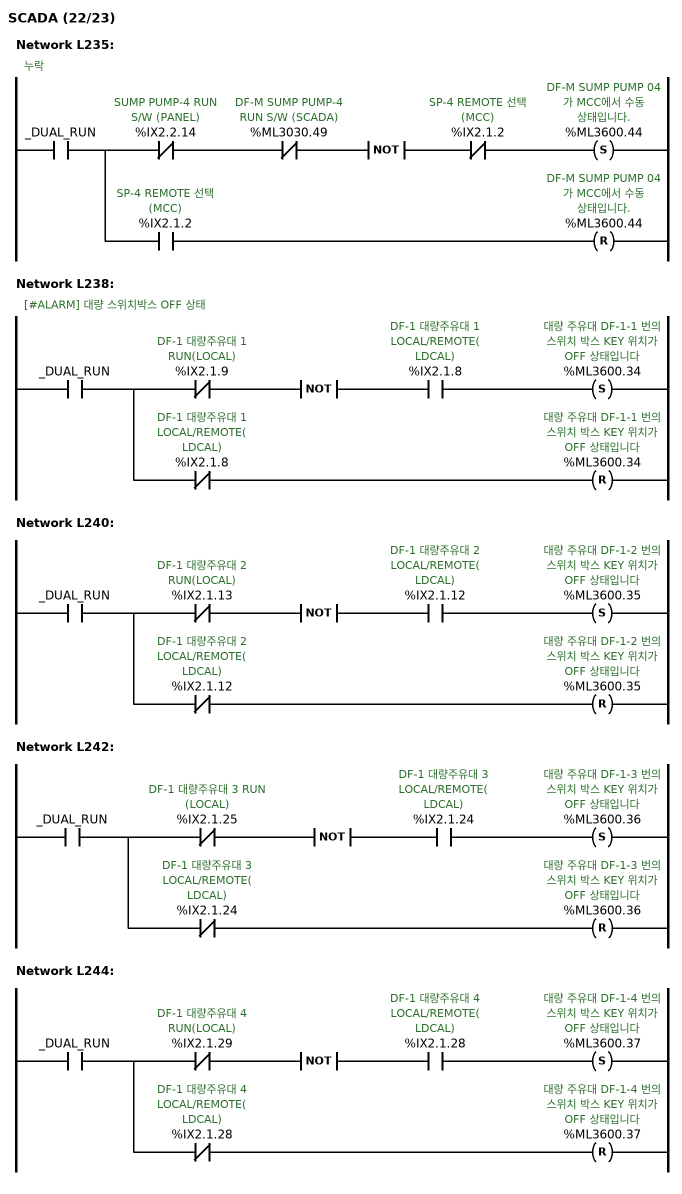
(* [picture p72: SCADA rungs L235-L244] *)
(* Rung L235 *)
IF NOT (_DUAL_RUN AND NOT %IX2.2.14 AND NOT %ML3030.49) AND NOT %IX2.1.2 THEN %ML3600.44 := TRUE; END_IF;
IF _DUAL_RUN AND %IX2.1.2 THEN %ML3600.44 := FALSE; END_IF;
(* 누락 *)
(* [#ALARM] 대량 스위치박스 OFF 상태 *)
(* Rung L238 *)
IF NOT (_DUAL_RUN AND NOT %IX2.1.9) AND %IX2.1.8 THEN %ML3600.34 := TRUE; END_IF;
IF _DUAL_RUN AND NOT %IX2.1.8 THEN %ML3600.34 := FALSE; END_IF;
(* Rung L240 *)
IF NOT (_DUAL_RUN AND NOT %IX2.1.13) AND %IX2.1.12 THEN %ML3600.35 := TRUE; END_IF;
IF _DUAL_RUN AND NOT %IX2.1.12 THEN %ML3600.35 := FALSE; END_IF;
(* Rung L242 *)
IF NOT (_DUAL_RUN AND NOT %IX2.1.25) AND %IX2.1.24 THEN %ML3600.36 := TRUE; END_IF;
IF _DUAL_RUN AND NOT %IX2.1.24 THEN %ML3600.36 := FALSE; END_IF;
(* Rung L244 *)
IF NOT (_DUAL_RUN AND NOT %IX2.1.29) AND %IX2.1.28 THEN %ML3600.37 := TRUE; END_IF;
IF _DUAL_RUN AND NOT %IX2.1.28 THEN %ML3600.37 := FALSE; END_IF;

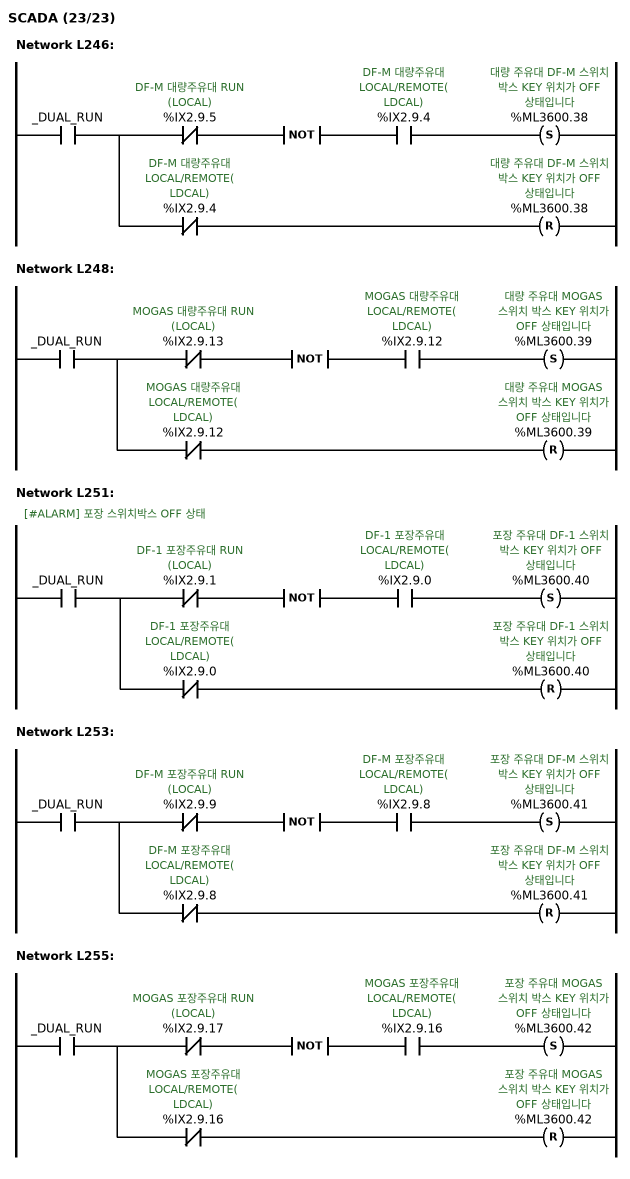
(* Rung L246 *)
IF NOT (_DUAL_RUN AND NOT %IX2.9.5) AND %IX2.9.4 THEN %ML3600.38 := TRUE; END_IF;
IF _DUAL_RUN AND NOT %IX2.9.4 THEN %ML3600.38 := FALSE; END_IF;
(* Rung L248 *)
IF NOT (_DUAL_RUN AND NOT %IX2.9.13) AND %IX2.9.12 THEN %ML3600.39 := TRUE; END_IF;
IF _DUAL_RUN AND NOT %IX2.9.12 THEN %ML3600.39 := FALSE; END_IF;
(* [#ALARM] 포장 스위치박스 OFF 상태 *)
(* Rung L251 *)
IF NOT (_DUAL_RUN AND NOT %IX2.9.1) AND %IX2.9.0 THEN %ML3600.40 := TRUE; END_IF;
IF _DUAL_RUN AND NOT %IX2.9.0 THEN %ML3600.40 := FALSE; END_IF;
(* Rung L253 *)
IF NOT (_DUAL_RUN AND NOT %IX2.9.9) AND %IX2.9.8 THEN %ML3600.41 := TRUE; END_IF;
IF _DUAL_RUN AND NOT %IX2.9.8 THEN %ML3600.41 := FALSE; END_IF;
(* Rung L255 *)
IF NOT (_DUAL_RUN AND NOT %IX2.9.17) AND %IX2.9.16 THEN %ML3600.42 := TRUE; END_IF;
IF _DUAL_RUN AND NOT %IX2.9.16 THEN %ML3600.42 := FALSE; END_IF;
END_PROGRAM

PROGRAM OUT (* task: 스캔 프로그램 *)
VAR
    D10 : BOOL;
    D1000 : BOOL;
    H16 : BOOL;
    INST : FF;
END_VAR
VAR
    _t1 : BOOL;
    _t2 : BOOL;
    _t3 : BOOL;
    _t4 : BOOL;
    _t5 : BOOL;
    _t6 : BOOL;
    _t7 : BOOL;
    _t8 : BOOL;
    _t9 : BOOL;
    _t10 : BOOL;
    _t11 : BOOL;
    _t12 : BOOL;
END_VAR

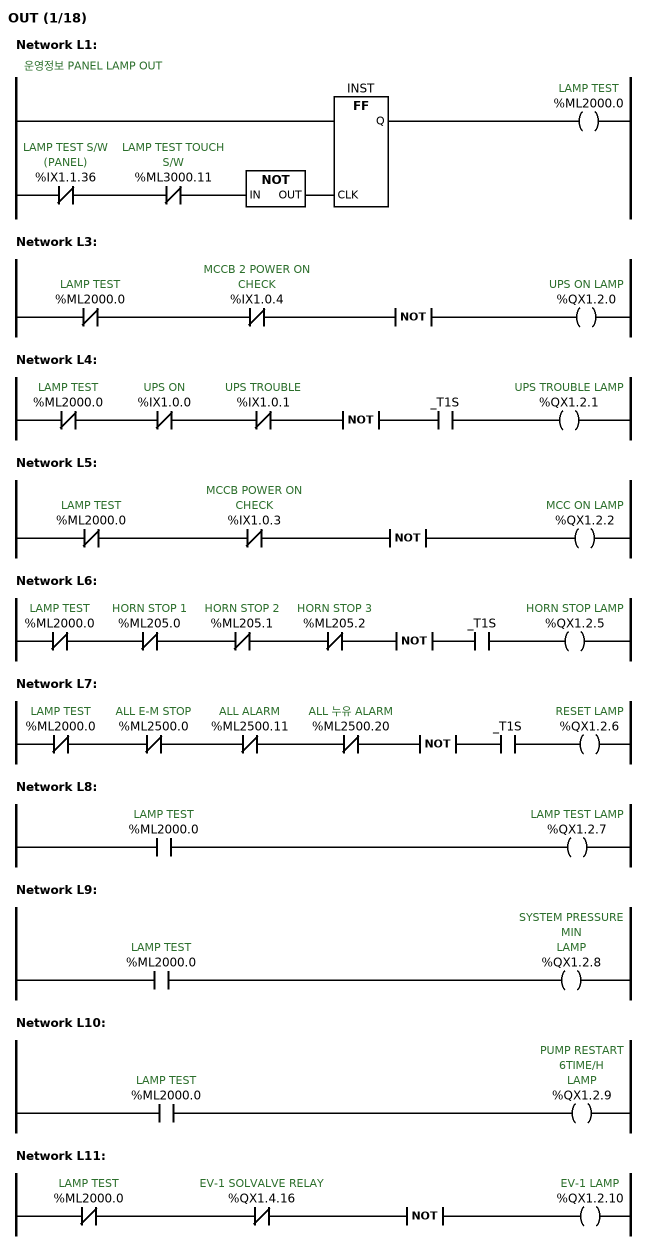
(* 운영정보 PANEL LAMP OUT *)
(* Rung L1 *)
INST(CLK := NOT (NOT %IX1.1.36 AND NOT %ML3000.11));
%ML2000.0 := INST.Q;
(* Rung L3 *)
%QX1.2.0 := NOT (NOT %ML2000.0 AND NOT %IX1.0.4);
(* Rung L4 *)
%QX1.2.1 := NOT (NOT %ML2000.0 AND NOT %IX1.0.0 AND NOT %IX1.0.1) AND _T1S;
(* Rung L5 *)
%QX1.2.2 := NOT (NOT %ML2000.0 AND NOT %IX1.0.3);
(* Rung L6 *)
%QX1.2.5 := NOT (NOT %ML2000.0 AND NOT %ML205.0 AND NOT %ML205.1 AND NOT %ML205.2) AND _T1S;
(* Rung L7 *)
%QX1.2.6 := NOT (NOT %ML2000.0 AND NOT %ML2500.0 AND NOT %ML2500.11 AND NOT %ML2500.20) AND _T1S;
(* Rung L8 *)
%QX1.2.7 := %ML2000.0;
(* Rung L9 *)
%QX1.2.8 := %ML2000.0;
(* Rung L10 *)
%QX1.2.9 := %ML2000.0;
(* Rung L11 *)
%QX1.2.10 := NOT (NOT %ML2000.0 AND NOT %QX1.4.16);

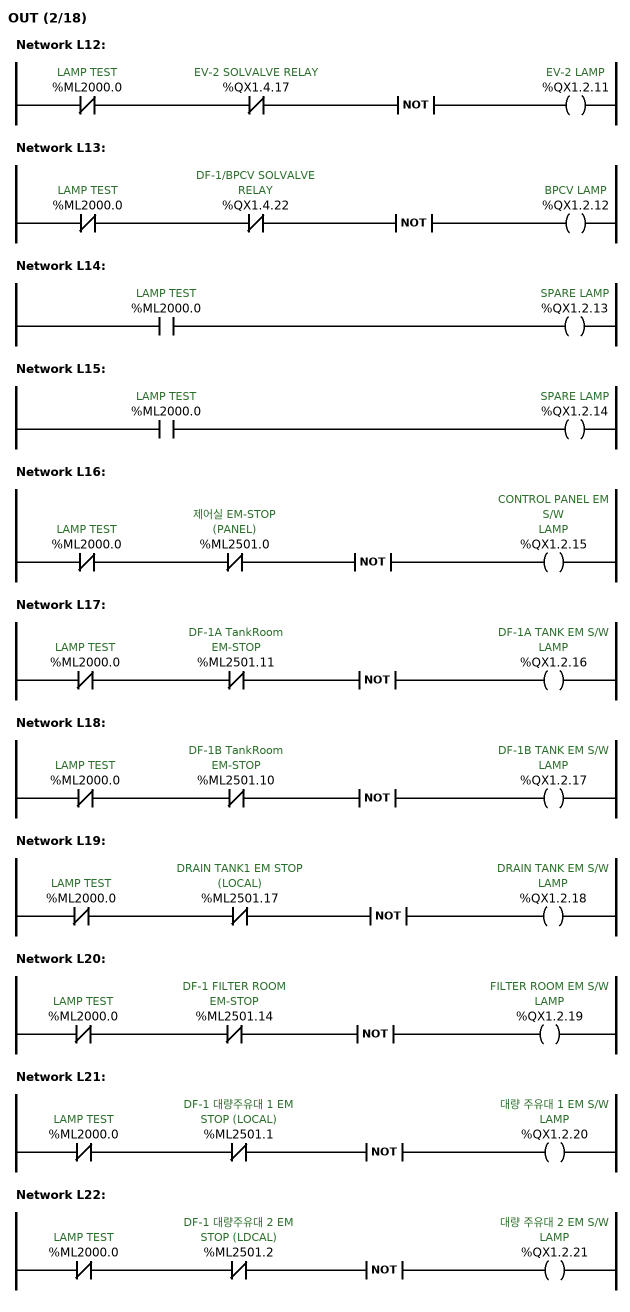
(* Rung L12 *)
%QX1.2.11 := NOT (NOT %ML2000.0 AND NOT %QX1.4.17);
(* Rung L13 *)
%QX1.2.12 := NOT (NOT %ML2000.0 AND NOT %QX1.4.22);
(* Rung L14 *)
%QX1.2.13 := %ML2000.0;
(* Rung L15 *)
%QX1.2.14 := %ML2000.0;
(* Rung L16 *)
%QX1.2.15 := NOT (NOT %ML2000.0 AND NOT %ML2501.0);
(* Rung L17 *)
%QX1.2.16 := NOT (NOT %ML2000.0 AND NOT %ML2501.11);
(* Rung L18 *)
%QX1.2.17 := NOT (NOT %ML2000.0 AND NOT %ML2501.10);
(* Rung L19 *)
%QX1.2.18 := NOT (NOT %ML2000.0 AND NOT %ML2501.17);
(* Rung L20 *)
%QX1.2.19 := NOT (NOT %ML2000.0 AND NOT %ML2501.14);
(* Rung L21 *)
%QX1.2.20 := NOT (NOT %ML2000.0 AND NOT %ML2501.1);
(* Rung L22 *)
%QX1.2.21 := NOT (NOT %ML2000.0 AND NOT %ML2501.2);

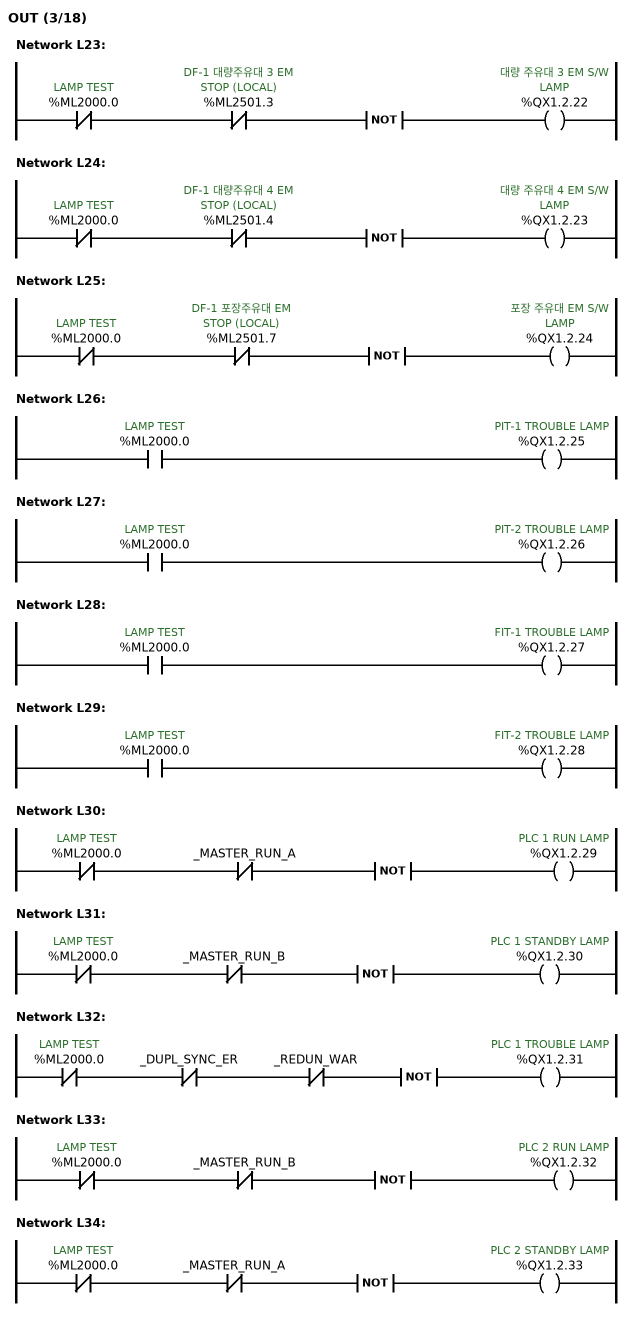
(* Rung L23 *)
%QX1.2.22 := NOT (NOT %ML2000.0 AND NOT %ML2501.3);
(* Rung L24 *)
%QX1.2.23 := NOT (NOT %ML2000.0 AND NOT %ML2501.4);
(* Rung L25 *)
%QX1.2.24 := NOT (NOT %ML2000.0 AND NOT %ML2501.7);
(* Rung L26 *)
%QX1.2.25 := %ML2000.0;
(* Rung L27 *)
%QX1.2.26 := %ML2000.0;
(* Rung L28 *)
%QX1.2.27 := %ML2000.0;
(* Rung L29 *)
%QX1.2.28 := %ML2000.0;
(* Rung L30 *)
%QX1.2.29 := NOT (NOT %ML2000.0 AND NOT _MASTER_RUN_A);
(* Rung L31 *)
%QX1.2.30 := NOT (NOT %ML2000.0 AND NOT _MASTER_RUN_B);
(* Rung L32 *)
%QX1.2.31 := NOT (NOT %ML2000.0 AND NOT _DUPL_SYNC_ER AND NOT _REDUN_WAR);
(* Rung L33 *)
%QX1.2.32 := NOT (NOT %ML2000.0 AND NOT _MASTER_RUN_B);
(* Rung L34 *)
%QX1.2.33 := NOT (NOT %ML2000.0 AND NOT _MASTER_RUN_A);

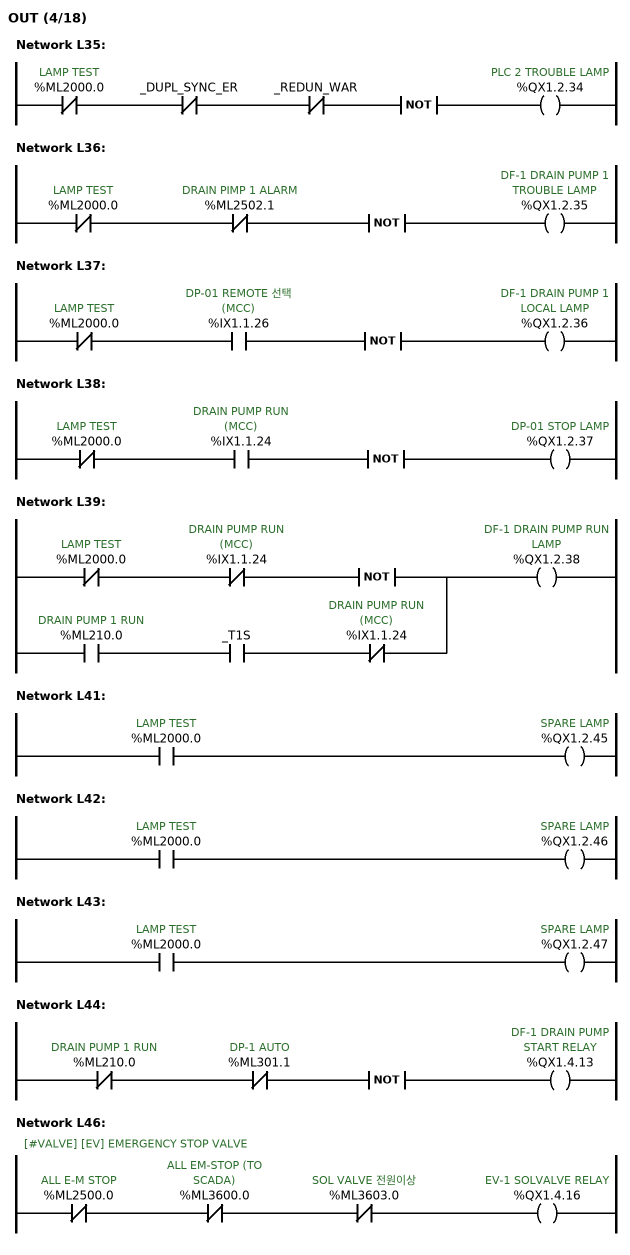
(* Rung L35 *)
%QX1.2.34 := NOT (NOT %ML2000.0 AND NOT _DUPL_SYNC_ER AND NOT _REDUN_WAR);
(* Rung L36 *)
%QX1.2.35 := NOT (NOT %ML2000.0 AND NOT %ML2502.1);
(* Rung L37 *)
%QX1.2.36 := NOT (NOT %ML2000.0 AND %IX1.1.26);
(* Rung L38 *)
%QX1.2.37 := NOT (NOT %ML2000.0 AND %IX1.1.24);
(* Rung L39 *)
%QX1.2.38 := NOT (NOT %ML2000.0 AND NOT %IX1.1.24) OR (%ML210.0 AND _T1S AND NOT %IX1.1.24);
(* Rung L41 *)
%QX1.2.45 := %ML2000.0;
(* Rung L42 *)
%QX1.2.46 := %ML2000.0;
(* Rung L43 *)
%QX1.2.47 := %ML2000.0;
(* Rung L44 *)
%QX1.4.13 := NOT (NOT %ML210.0 AND NOT %ML301.1);
(* [#VALVE] [EV] EMERGENCY STOP VALVE *)
(* Rung L46 *)
%QX1.4.16 := NOT %ML2500.0 AND NOT %ML3600.0 AND NOT %ML3603.0;

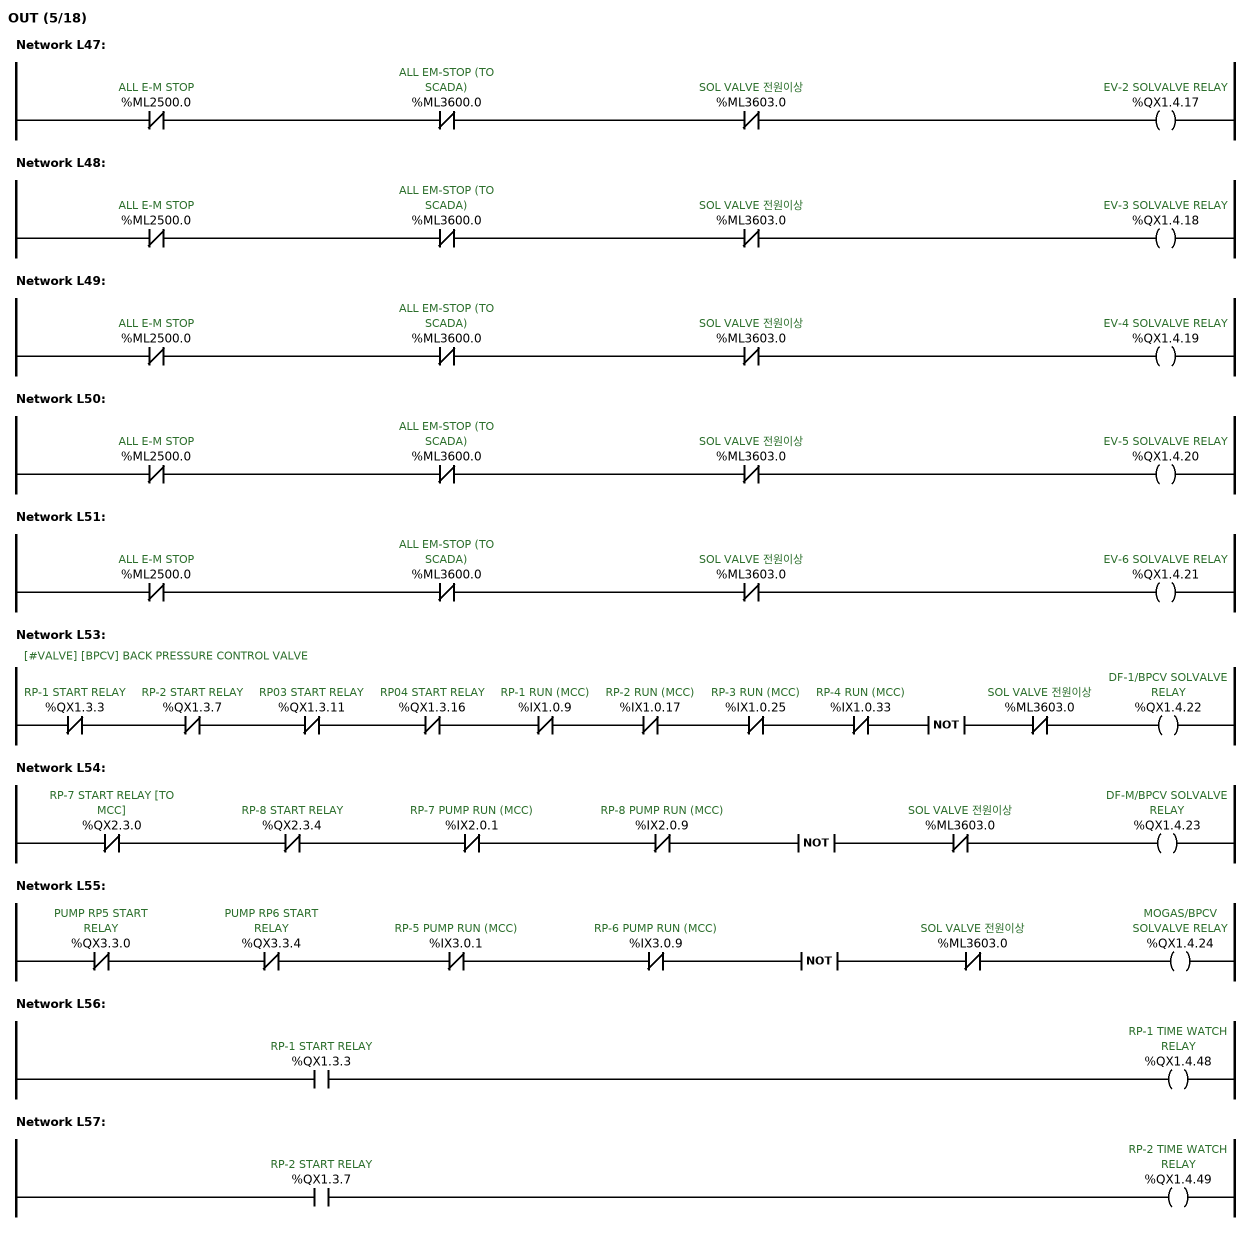
(* Rung L47 *)
%QX1.4.17 := NOT %ML2500.0 AND NOT %ML3600.0 AND NOT %ML3603.0;
(* Rung L48 *)
%QX1.4.18 := NOT %ML2500.0 AND NOT %ML3600.0 AND NOT %ML3603.0;
(* Rung L49 *)
%QX1.4.19 := NOT %ML2500.0 AND NOT %ML3600.0 AND NOT %ML3603.0;
(* Rung L50 *)
%QX1.4.20 := NOT %ML2500.0 AND NOT %ML3600.0 AND NOT %ML3603.0;
(* Rung L51 *)
%QX1.4.21 := NOT %ML2500.0 AND NOT %ML3600.0 AND NOT %ML3603.0;
(* [#VALVE] [BPCV] BACK PRESSURE CONTROL VALVE *)
(* Rung L53 *)
%QX1.4.22 := NOT (NOT %QX1.3.3 AND NOT %QX1.3.7 AND NOT %QX1.3.11 AND NOT %QX1.3.16 AND NOT %IX1.0.9 AND NOT %IX1.0.17 AND NOT %IX1.0.25 AND NOT %IX1.0.33) AND NOT %ML3603.0;
(* Rung L54 *)
%QX1.4.23 := NOT (NOT %QX2.3.0 AND NOT %QX2.3.4 AND NOT %IX2.0.1 AND NOT %IX2.0.9) AND NOT %ML3603.0;
(* Rung L55 *)
%QX1.4.24 := NOT (NOT %QX3.3.0 AND NOT %QX3.3.4 AND NOT %IX3.0.1 AND NOT %IX3.0.9) AND NOT %ML3603.0;
(* Rung L56 *)
%QX1.4.48 := %QX1.3.3;
(* Rung L57 *)
%QX1.4.49 := %QX1.3.7;

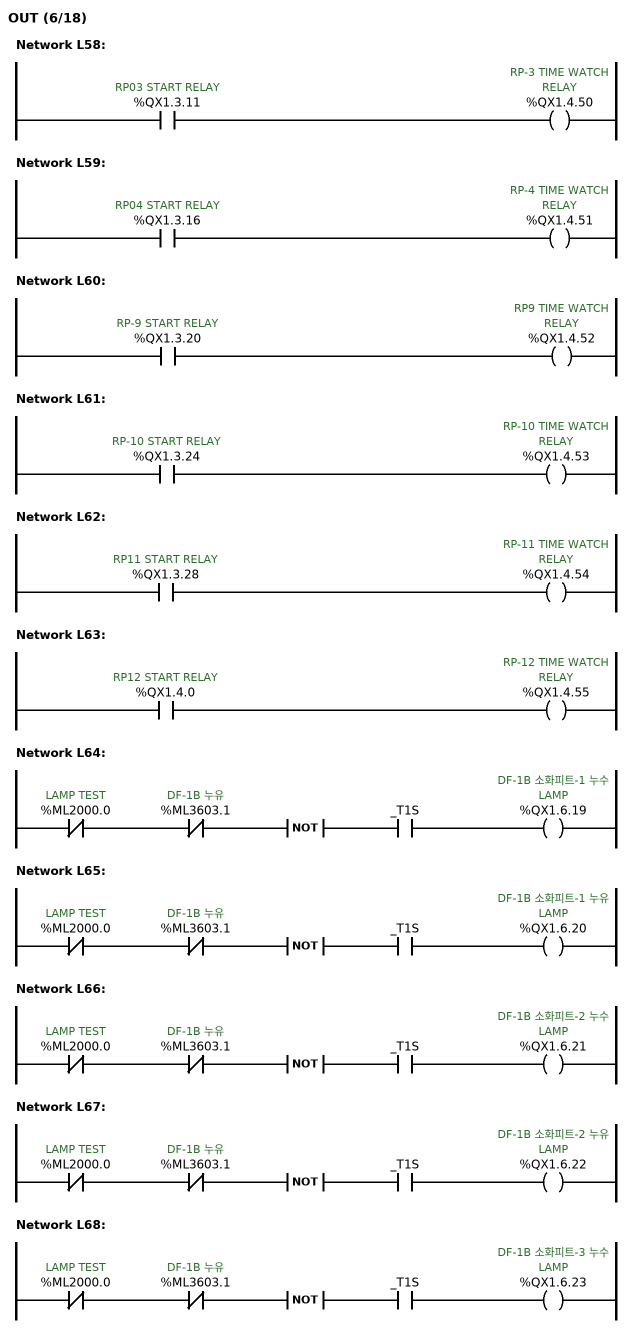
(* Rung L58 *)
%QX1.4.50 := %QX1.3.11;
(* Rung L59 *)
%QX1.4.51 := %QX1.3.16;
(* Rung L60 *)
%QX1.4.52 := %QX1.3.20;
(* Rung L61 *)
%QX1.4.53 := %QX1.3.24;
(* Rung L62 *)
%QX1.4.54 := %QX1.3.28;
(* Rung L63 *)
%QX1.4.55 := %QX1.4.0;
(* Rung L64 *)
%QX1.6.19 := NOT (NOT %ML2000.0 AND NOT %ML3603.1) AND _T1S;
(* Rung L65 *)
%QX1.6.20 := NOT (NOT %ML2000.0 AND NOT %ML3603.1) AND _T1S;
(* Rung L66 *)
%QX1.6.21 := NOT (NOT %ML2000.0 AND NOT %ML3603.1) AND _T1S;
(* Rung L67 *)
%QX1.6.22 := NOT (NOT %ML2000.0 AND NOT %ML3603.1) AND _T1S;
(* Rung L68 *)
%QX1.6.23 := NOT (NOT %ML2000.0 AND NOT %ML3603.1) AND _T1S;

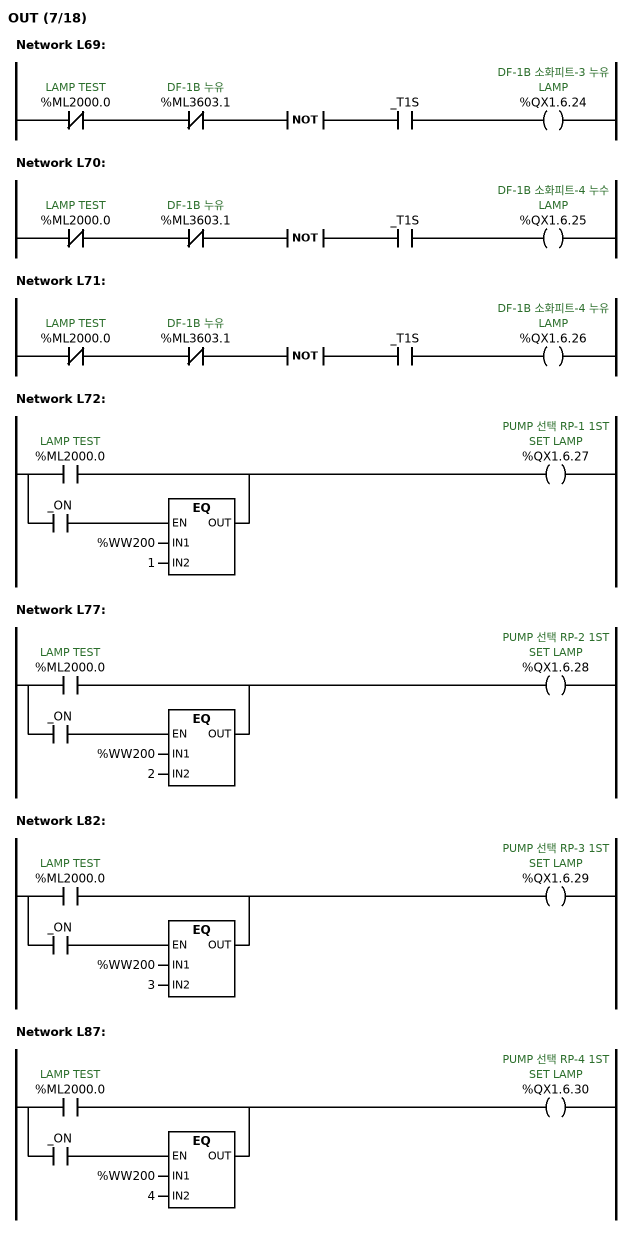
(* Rung L69 *)
%QX1.6.24 := NOT (NOT %ML2000.0 AND NOT %ML3603.1) AND _T1S;
(* Rung L70 *)
%QX1.6.25 := NOT (NOT %ML2000.0 AND NOT %ML3603.1) AND _T1S;
(* Rung L71 *)
%QX1.6.26 := NOT (NOT %ML2000.0 AND NOT %ML3603.1) AND _T1S;
(* Rung L72 *)
IF _ON THEN _t1 := %WW200 = 1; END_IF;
%QX1.6.27 := %ML2000.0 OR _t1;
(* Rung L77 *)
IF _ON THEN _t2 := %WW200 = 2; END_IF;
%QX1.6.28 := %ML2000.0 OR _t2;
(* Rung L82 *)
IF _ON THEN _t3 := %WW200 = 3; END_IF;
%QX1.6.29 := %ML2000.0 OR _t3;
(* Rung L87 *)
IF _ON THEN _t4 := %WW200 = 4; END_IF;
%QX1.6.30 := %ML2000.0 OR _t4;

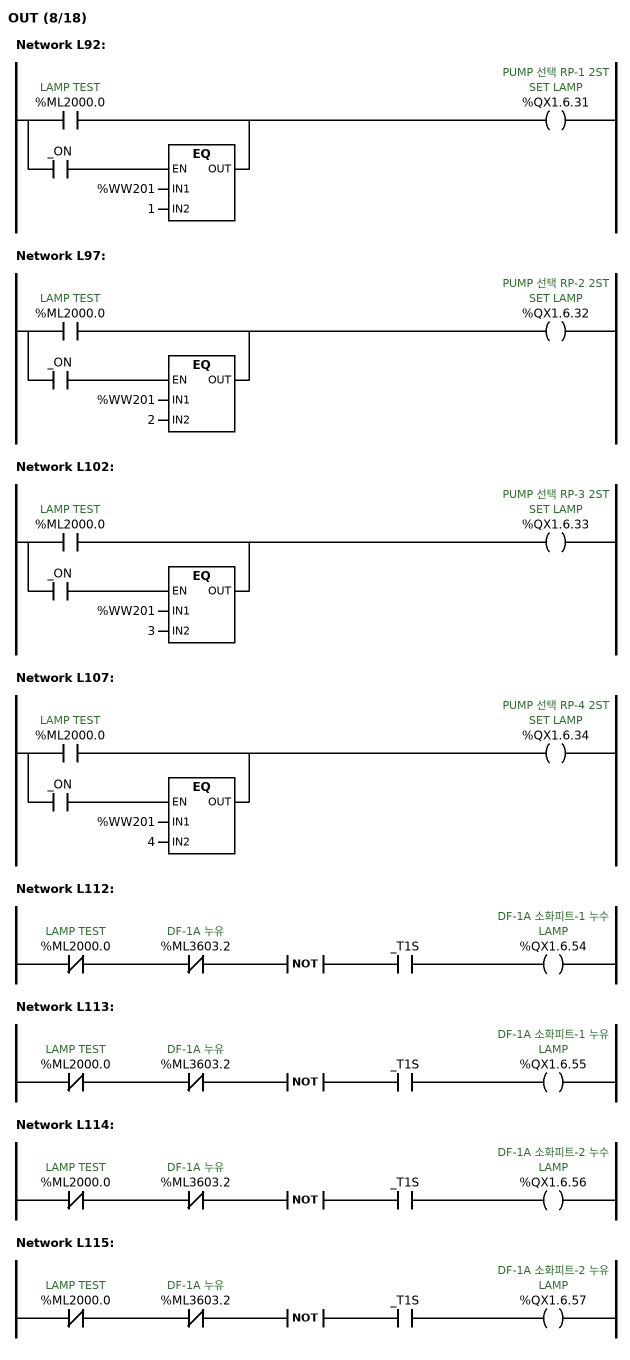
(* Rung L92 *)
IF _ON THEN _t5 := %WW201 = 1; END_IF;
%QX1.6.31 := %ML2000.0 OR _t5;
(* Rung L97 *)
IF _ON THEN _t6 := %WW201 = 2; END_IF;
%QX1.6.32 := %ML2000.0 OR _t6;
(* Rung L102 *)
IF _ON THEN _t7 := %WW201 = 3; END_IF;
%QX1.6.33 := %ML2000.0 OR _t7;
(* Rung L107 *)
IF _ON THEN _t8 := %WW201 = 4; END_IF;
%QX1.6.34 := %ML2000.0 OR _t8;
(* Rung L112 *)
%QX1.6.54 := NOT (NOT %ML2000.0 AND NOT %ML3603.2) AND _T1S;
(* Rung L113 *)
%QX1.6.55 := NOT (NOT %ML2000.0 AND NOT %ML3603.2) AND _T1S;
(* Rung L114 *)
%QX1.6.56 := NOT (NOT %ML2000.0 AND NOT %ML3603.2) AND _T1S;
(* Rung L115 *)
%QX1.6.57 := NOT (NOT %ML2000.0 AND NOT %ML3603.2) AND _T1S;

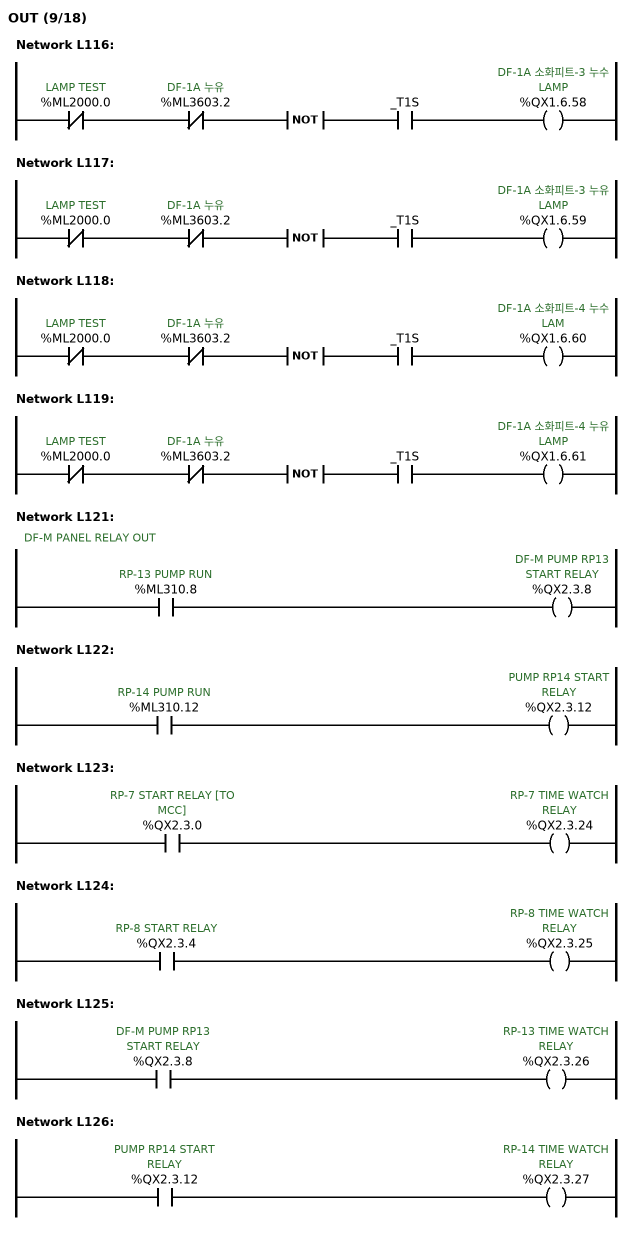
(* Rung L116 *)
%QX1.6.58 := NOT (NOT %ML2000.0 AND NOT %ML3603.2) AND _T1S;
(* Rung L117 *)
%QX1.6.59 := NOT (NOT %ML2000.0 AND NOT %ML3603.2) AND _T1S;
(* Rung L118 *)
%QX1.6.60 := NOT (NOT %ML2000.0 AND NOT %ML3603.2) AND _T1S;
(* Rung L119 *)
%QX1.6.61 := NOT (NOT %ML2000.0 AND NOT %ML3603.2) AND _T1S;
(* DF-M PANEL RELAY OUT *)
(* Rung L121 *)
%QX2.3.8 := %ML310.8;
(* Rung L122 *)
%QX2.3.12 := %ML310.12;
(* Rung L123 *)
%QX2.3.24 := %QX2.3.0;
(* Rung L124 *)
%QX2.3.25 := %QX2.3.4;
(* Rung L125 *)
%QX2.3.26 := %QX2.3.8;
(* Rung L126 *)
%QX2.3.27 := %QX2.3.12;

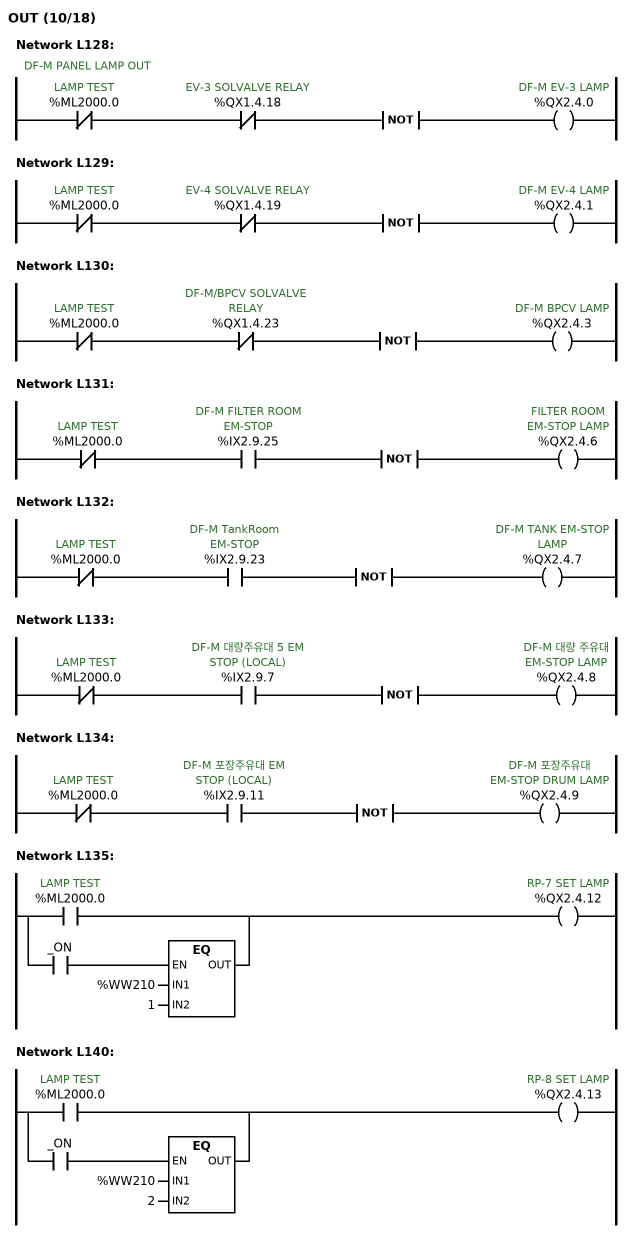
(* DF-M PANEL LAMP OUT *)
(* Rung L128 *)
%QX2.4.0 := NOT (NOT %ML2000.0 AND NOT %QX1.4.18);
(* Rung L129 *)
%QX2.4.1 := NOT (NOT %ML2000.0 AND NOT %QX1.4.19);
(* Rung L130 *)
%QX2.4.3 := NOT (NOT %ML2000.0 AND NOT %QX1.4.23);
(* Rung L131 *)
%QX2.4.6 := NOT (NOT %ML2000.0 AND %IX2.9.25);
(* Rung L132 *)
%QX2.4.7 := NOT (NOT %ML2000.0 AND %IX2.9.23);
(* Rung L133 *)
%QX2.4.8 := NOT (NOT %ML2000.0 AND %IX2.9.7);
(* Rung L134 *)
%QX2.4.9 := NOT (NOT %ML2000.0 AND %IX2.9.11);
(* Rung L135 *)
IF _ON THEN _t9 := %WW210 = 1; END_IF;
%QX2.4.12 := %ML2000.0 OR _t9;
(* Rung L140 *)
IF _ON THEN _t10 := %WW210 = 2; END_IF;
%QX2.4.13 := %ML2000.0 OR _t10;

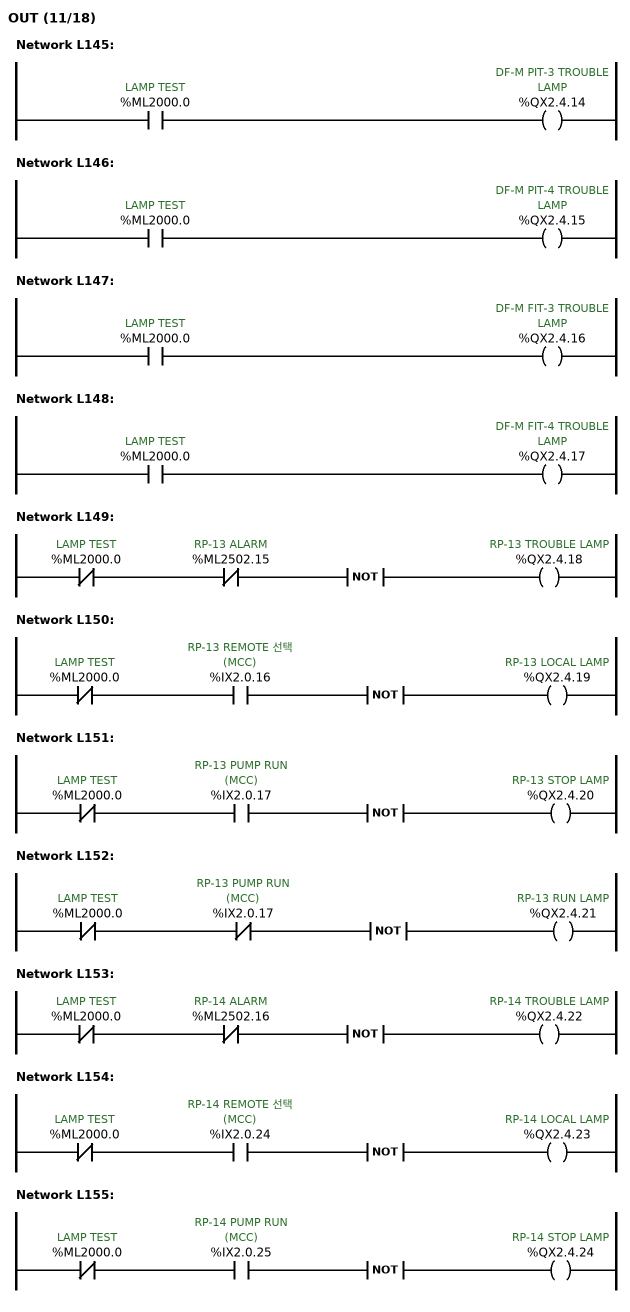
(* Rung L145 *)
%QX2.4.14 := %ML2000.0;
(* Rung L146 *)
%QX2.4.15 := %ML2000.0;
(* Rung L147 *)
%QX2.4.16 := %ML2000.0;
(* Rung L148 *)
%QX2.4.17 := %ML2000.0;
(* Rung L149 *)
%QX2.4.18 := NOT (NOT %ML2000.0 AND NOT %ML2502.15);
(* Rung L150 *)
%QX2.4.19 := NOT (NOT %ML2000.0 AND %IX2.0.16);
(* Rung L151 *)
%QX2.4.20 := NOT (NOT %ML2000.0 AND %IX2.0.17);
(* Rung L152 *)
%QX2.4.21 := NOT (NOT %ML2000.0 AND NOT %IX2.0.17);
(* Rung L153 *)
%QX2.4.22 := NOT (NOT %ML2000.0 AND NOT %ML2502.16);
(* Rung L154 *)
%QX2.4.23 := NOT (NOT %ML2000.0 AND %IX2.0.24);
(* Rung L155 *)
%QX2.4.24 := NOT (NOT %ML2000.0 AND %IX2.0.25);

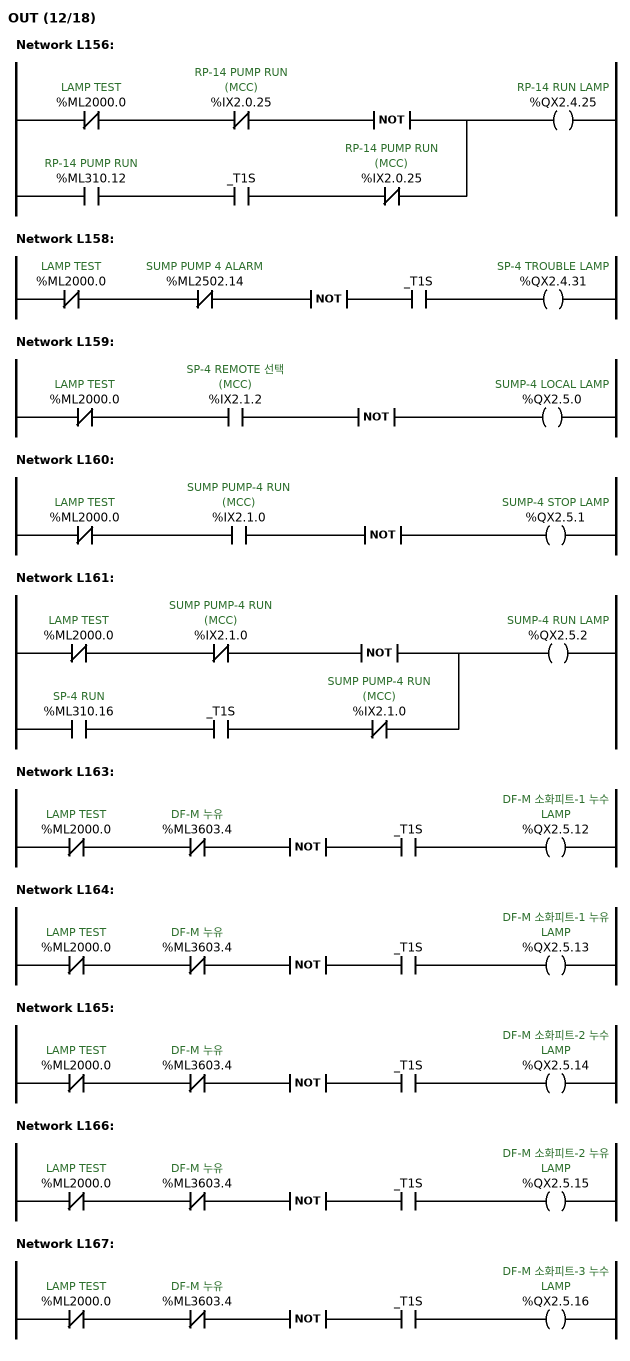
(* Rung L156 *)
%QX2.4.25 := NOT (NOT %ML2000.0 AND NOT %IX2.0.25) OR (%ML310.12 AND _T1S AND NOT %IX2.0.25);
(* Rung L158 *)
%QX2.4.31 := NOT (NOT %ML2000.0 AND NOT %ML2502.14) AND _T1S;
(* Rung L159 *)
%QX2.5.0 := NOT (NOT %ML2000.0 AND %IX2.1.2);
(* Rung L160 *)
%QX2.5.1 := NOT (NOT %ML2000.0 AND %IX2.1.0);
(* Rung L161 *)
%QX2.5.2 := NOT (NOT %ML2000.0 AND NOT %IX2.1.0) OR (%ML310.16 AND _T1S AND NOT %IX2.1.0);
(* Rung L163 *)
%QX2.5.12 := NOT (NOT %ML2000.0 AND NOT %ML3603.4) AND _T1S;
(* Rung L164 *)
%QX2.5.13 := NOT (NOT %ML2000.0 AND NOT %ML3603.4) AND _T1S;
(* Rung L165 *)
%QX2.5.14 := NOT (NOT %ML2000.0 AND NOT %ML3603.4) AND _T1S;
(* Rung L166 *)
%QX2.5.15 := NOT (NOT %ML2000.0 AND NOT %ML3603.4) AND _T1S;
(* Rung L167 *)
%QX2.5.16 := NOT (NOT %ML2000.0 AND NOT %ML3603.4) AND _T1S;

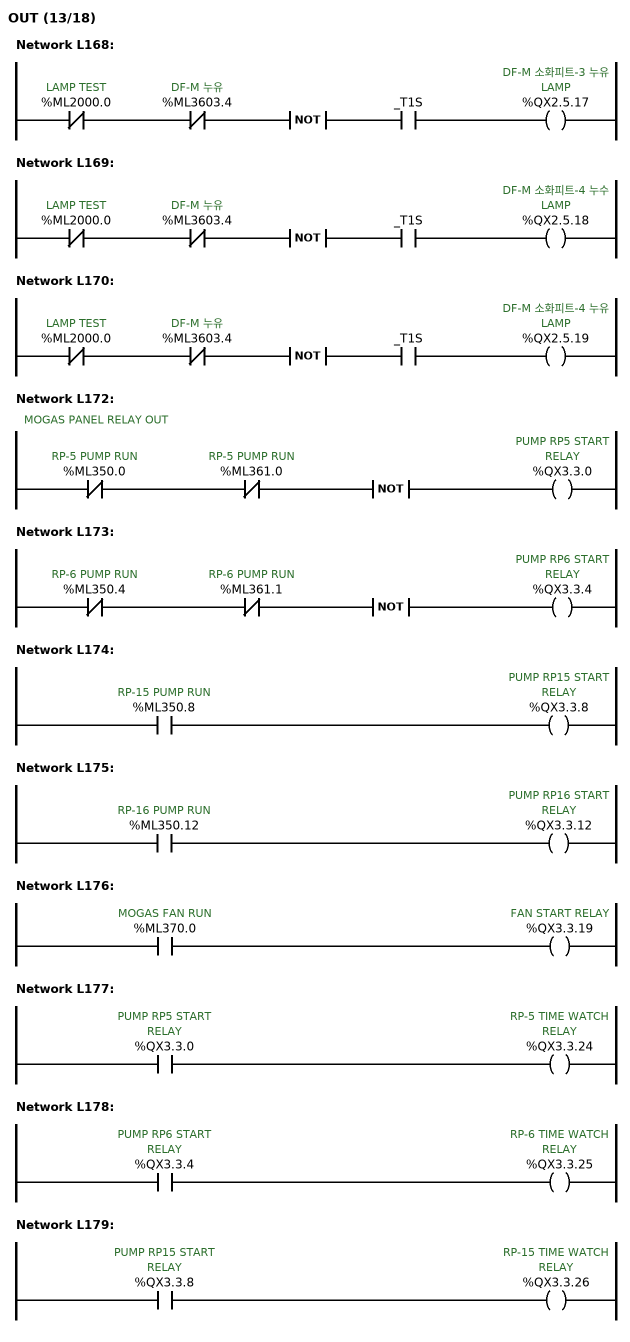
(* Rung L168 *)
%QX2.5.17 := NOT (NOT %ML2000.0 AND NOT %ML3603.4) AND _T1S;
(* Rung L169 *)
%QX2.5.18 := NOT (NOT %ML2000.0 AND NOT %ML3603.4) AND _T1S;
(* Rung L170 *)
%QX2.5.19 := NOT (NOT %ML2000.0 AND NOT %ML3603.4) AND _T1S;
(* MOGAS PANEL RELAY OUT *)
(* Rung L172 *)
%QX3.3.0 := NOT (NOT %ML350.0 AND NOT %ML361.0);
(* Rung L173 *)
%QX3.3.4 := NOT (NOT %ML350.4 AND NOT %ML361.1);
(* Rung L174 *)
%QX3.3.8 := %ML350.8;
(* Rung L175 *)
%QX3.3.12 := %ML350.12;
(* Rung L176 *)
%QX3.3.19 := %ML370.0;
(* Rung L177 *)
%QX3.3.24 := %QX3.3.0;
(* Rung L178 *)
%QX3.3.25 := %QX3.3.4;
(* Rung L179 *)
%QX3.3.26 := %QX3.3.8;

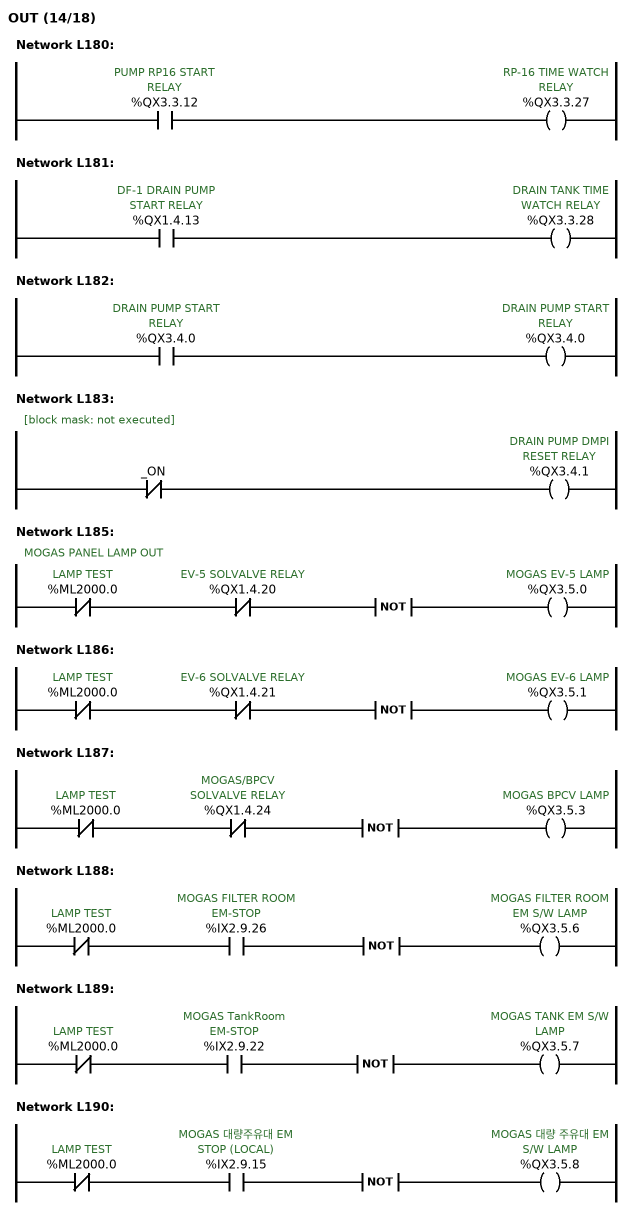
(* Rung L180 *)
%QX3.3.27 := %QX3.3.12;
(* Rung L181 *)
%QX3.3.28 := %QX1.4.13;
(* Rung L182 *)
%QX3.4.0 := %QX3.4.0;
(* Rung L183 is block-masked: not executed *)
// %QX3.4.1 := NOT _ON;
(* MOGAS PANEL LAMP OUT *)
(* Rung L185 *)
%QX3.5.0 := NOT (NOT %ML2000.0 AND NOT %QX1.4.20);
(* Rung L186 *)
%QX3.5.1 := NOT (NOT %ML2000.0 AND NOT %QX1.4.21);
(* Rung L187 *)
%QX3.5.3 := NOT (NOT %ML2000.0 AND NOT %QX1.4.24);
(* Rung L188 *)
%QX3.5.6 := NOT (NOT %ML2000.0 AND %IX2.9.26);
(* Rung L189 *)
%QX3.5.7 := NOT (NOT %ML2000.0 AND %IX2.9.22);
(* Rung L190 *)
%QX3.5.8 := NOT (NOT %ML2000.0 AND %IX2.9.15);

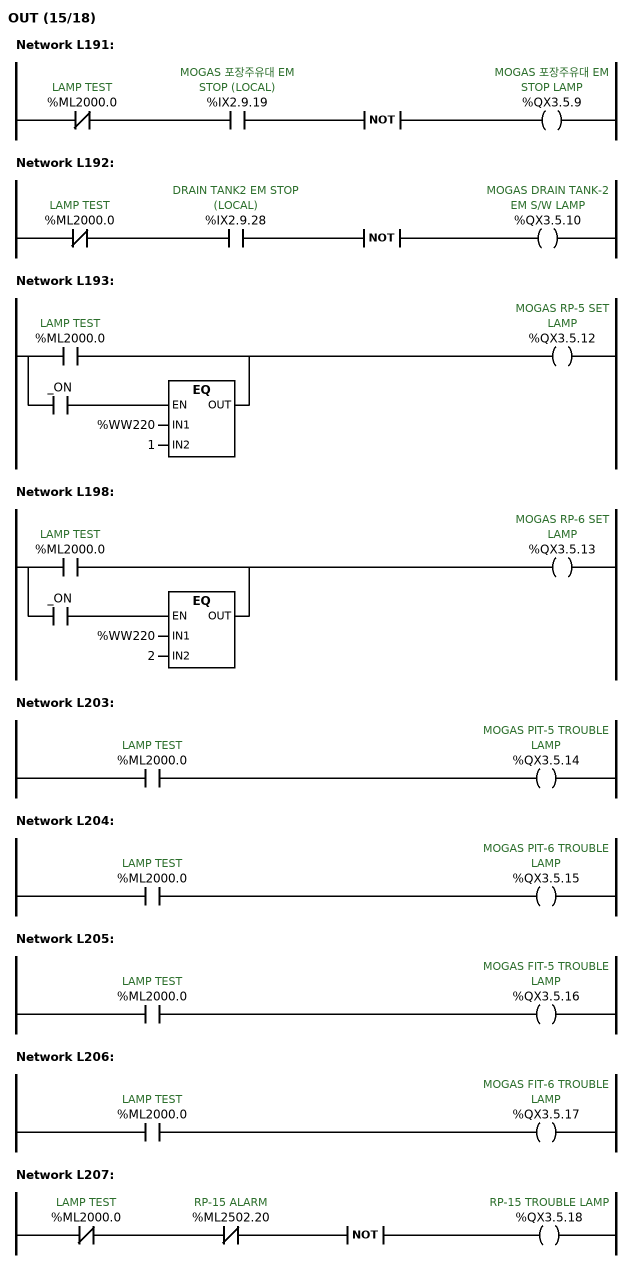
(* Rung L191 *)
%QX3.5.9 := NOT (NOT %ML2000.0 AND %IX2.9.19);
(* Rung L192 *)
%QX3.5.10 := NOT (NOT %ML2000.0 AND %IX2.9.28);
(* Rung L193 *)
IF _ON THEN _t11 := %WW220 = 1; END_IF;
%QX3.5.12 := %ML2000.0 OR _t11;
(* Rung L198 *)
IF _ON THEN _t12 := %WW220 = 2; END_IF;
%QX3.5.13 := %ML2000.0 OR _t12;
(* Rung L203 *)
%QX3.5.14 := %ML2000.0;
(* Rung L204 *)
%QX3.5.15 := %ML2000.0;
(* Rung L205 *)
%QX3.5.16 := %ML2000.0;
(* Rung L206 *)
%QX3.5.17 := %ML2000.0;
(* Rung L207 *)
%QX3.5.18 := NOT (NOT %ML2000.0 AND NOT %ML2502.20);

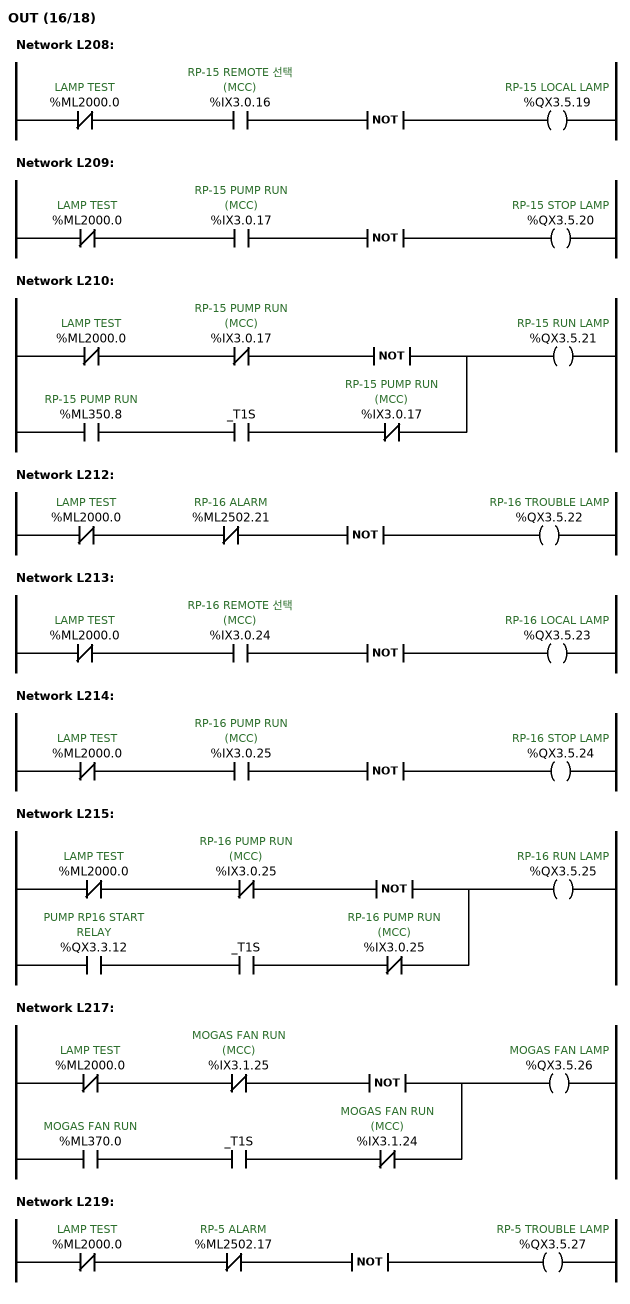
(* Rung L208 *)
%QX3.5.19 := NOT (NOT %ML2000.0 AND %IX3.0.16);
(* Rung L209 *)
%QX3.5.20 := NOT (NOT %ML2000.0 AND %IX3.0.17);
(* Rung L210 *)
%QX3.5.21 := NOT (NOT %ML2000.0 AND NOT %IX3.0.17) OR (%ML350.8 AND _T1S AND NOT %IX3.0.17);
(* Rung L212 *)
%QX3.5.22 := NOT (NOT %ML2000.0 AND NOT %ML2502.21);
(* Rung L213 *)
%QX3.5.23 := NOT (NOT %ML2000.0 AND %IX3.0.24);
(* Rung L214 *)
%QX3.5.24 := NOT (NOT %ML2000.0 AND %IX3.0.25);
(* Rung L215 *)
%QX3.5.25 := NOT (NOT %ML2000.0 AND NOT %IX3.0.25) OR (%QX3.3.12 AND _T1S AND NOT %IX3.0.25);
(* Rung L217 *)
%QX3.5.26 := NOT (NOT %ML2000.0 AND NOT %IX3.1.25) OR (%ML370.0 AND _T1S AND NOT %IX3.1.24);
(* Rung L219 *)
%QX3.5.27 := NOT (NOT %ML2000.0 AND NOT %ML2502.17);

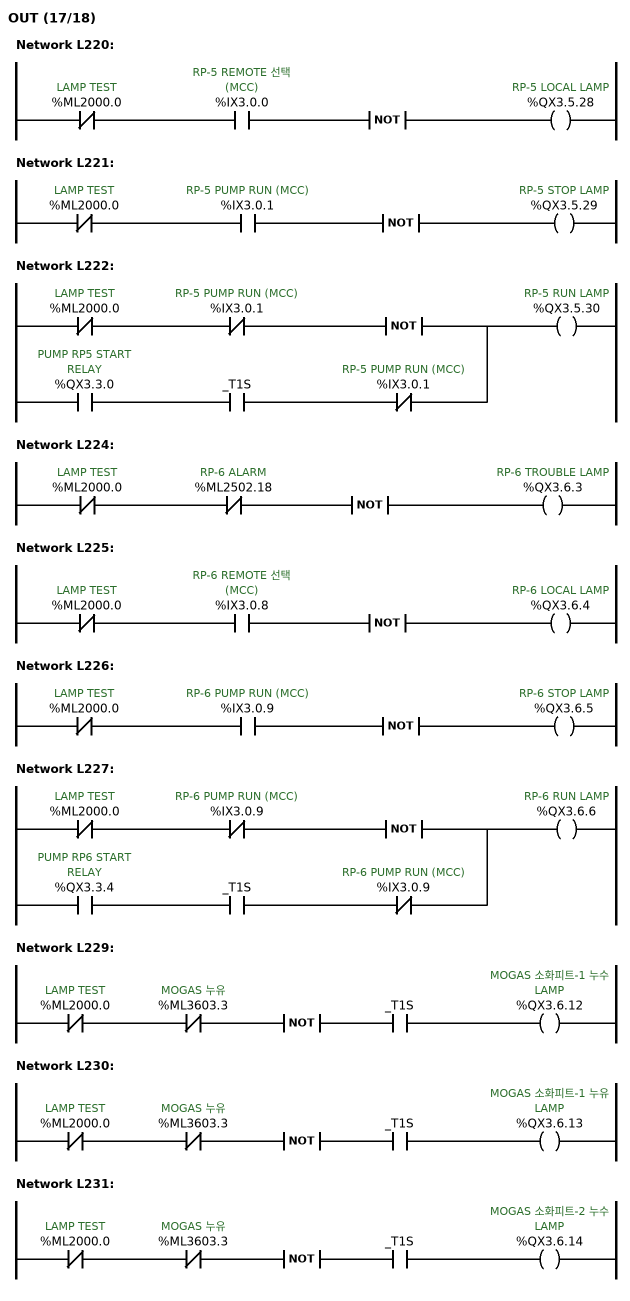
(* Rung L220 *)
%QX3.5.28 := NOT (NOT %ML2000.0 AND %IX3.0.0);
(* Rung L221 *)
%QX3.5.29 := NOT (NOT %ML2000.0 AND %IX3.0.1);
(* Rung L222 *)
%QX3.5.30 := NOT (NOT %ML2000.0 AND NOT %IX3.0.1) OR (%QX3.3.0 AND _T1S AND NOT %IX3.0.1);
(* Rung L224 *)
%QX3.6.3 := NOT (NOT %ML2000.0 AND NOT %ML2502.18);
(* Rung L225 *)
%QX3.6.4 := NOT (NOT %ML2000.0 AND %IX3.0.8);
(* Rung L226 *)
%QX3.6.5 := NOT (NOT %ML2000.0 AND %IX3.0.9);
(* Rung L227 *)
%QX3.6.6 := NOT (NOT %ML2000.0 AND NOT %IX3.0.9) OR (%QX3.3.4 AND _T1S AND NOT %IX3.0.9);
(* Rung L229 *)
%QX3.6.12 := NOT (NOT %ML2000.0 AND NOT %ML3603.3) AND _T1S;
(* Rung L230 *)
%QX3.6.13 := NOT (NOT %ML2000.0 AND NOT %ML3603.3) AND _T1S;
(* Rung L231 *)
%QX3.6.14 := NOT (NOT %ML2000.0 AND NOT %ML3603.3) AND _T1S;

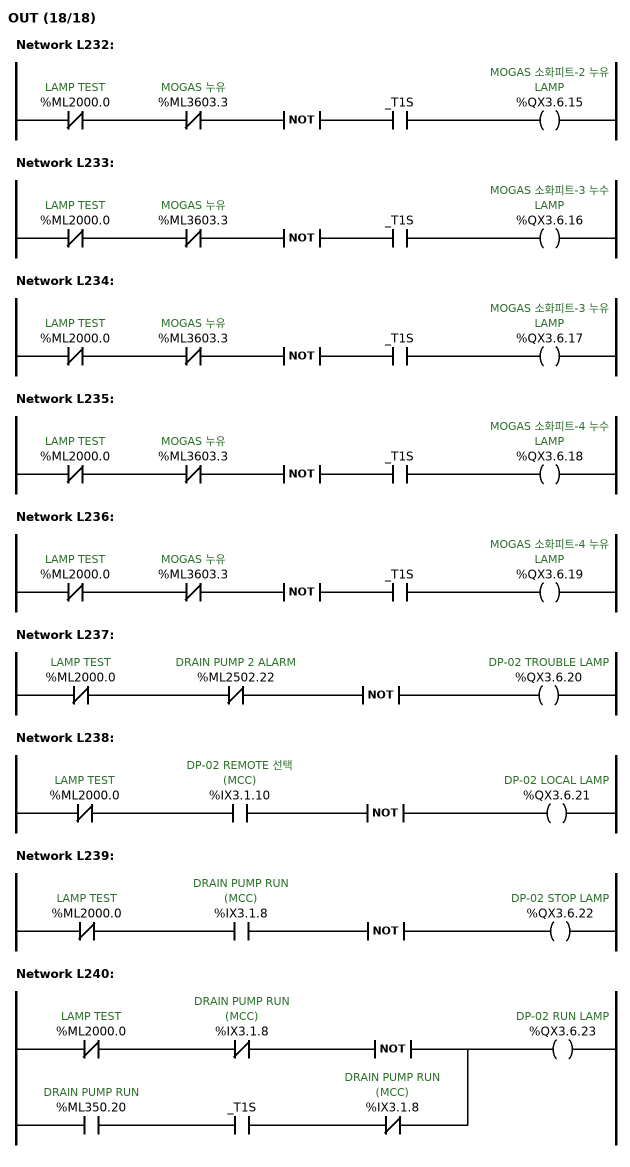
(* Rung L232 *)
%QX3.6.15 := NOT (NOT %ML2000.0 AND NOT %ML3603.3) AND _T1S;
(* Rung L233 *)
%QX3.6.16 := NOT (NOT %ML2000.0 AND NOT %ML3603.3) AND _T1S;
(* Rung L234 *)
%QX3.6.17 := NOT (NOT %ML2000.0 AND NOT %ML3603.3) AND _T1S;
(* Rung L235 *)
%QX3.6.18 := NOT (NOT %ML2000.0 AND NOT %ML3603.3) AND _T1S;
(* Rung L236 *)
%QX3.6.19 := NOT (NOT %ML2000.0 AND NOT %ML3603.3) AND _T1S;
(* Rung L237 *)
%QX3.6.20 := NOT (NOT %ML2000.0 AND NOT %ML2502.22);
(* Rung L238 *)
%QX3.6.21 := NOT (NOT %ML2000.0 AND %IX3.1.10);
(* Rung L239 *)
%QX3.6.22 := NOT (NOT %ML2000.0 AND %IX3.1.8);
(* Rung L240 *)
%QX3.6.23 := NOT (NOT %ML2000.0 AND NOT %IX3.1.8) OR (%ML350.20 AND _T1S AND NOT %IX3.1.8);
END_PROGRAM

PROGRAM ALARM (* task: 스캔 프로그램 *)

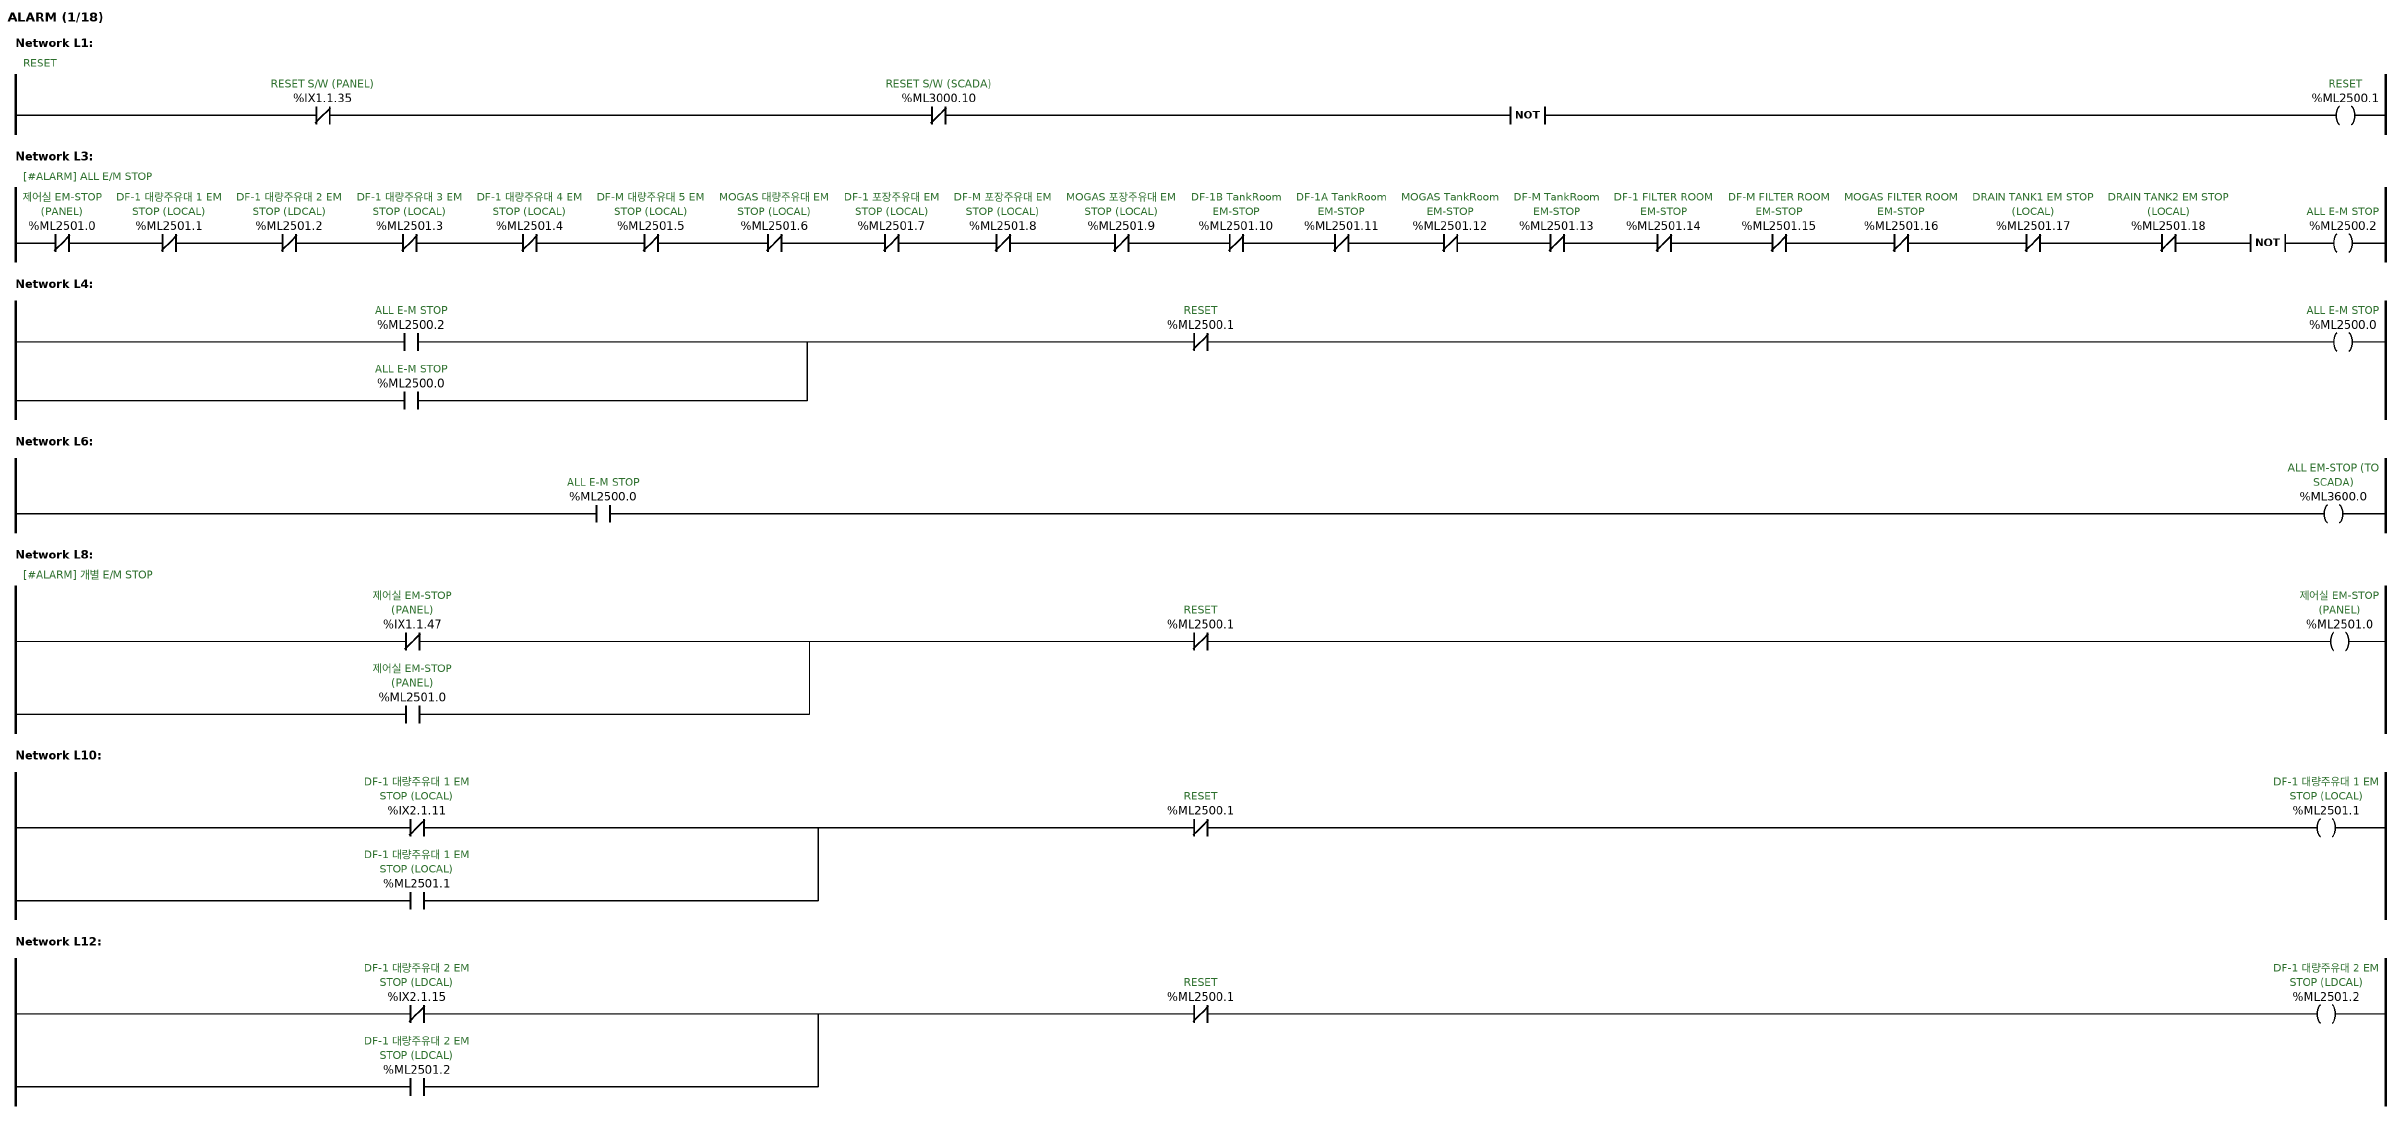
(* RESET *)
(* Rung L1 *)
%ML2500.1 := NOT (NOT %IX1.1.35 AND NOT %ML3000.10);
(* [#ALARM] ALL E/M STOP *)
(* Rung L3 *)
%ML2500.2 := NOT (NOT %ML2501.0 AND NOT %ML2501.1 AND NOT %ML2501.2 AND NOT %ML2501.3 AND NOT %ML2501.4 AND NOT %ML2501.5 AND NOT %ML2501.6 AND NOT %ML2501.7 AND NOT %ML2501.8 AND NOT %ML2501.9 AND NOT %ML2501.10 AND NOT %ML2501.11 AND NOT %ML2501.12 AND NOT %ML2501.13 AND NOT %ML2501.14 AND NOT %ML2501.15 AND NOT %ML2501.16 AND NOT %ML2501.17 AND NOT %ML2501.18);
(* Rung L4 *)
%ML2500.0 := (%ML2500.2 OR %ML2500.0) AND NOT %ML2500.1;
(* Rung L6 *)
%ML3600.0 := %ML2500.0;
(* [#ALARM] 개별 E/M STOP *)
(* Rung L8 *)
%ML2501.0 := (NOT %IX1.1.47 OR %ML2501.0) AND NOT %ML2500.1;
(* Rung L10 *)
%ML2501.1 := (NOT %IX2.1.11 OR %ML2501.1) AND NOT %ML2500.1;
(* Rung L12 *)
%ML2501.2 := (NOT %IX2.1.15 OR %ML2501.2) AND NOT %ML2500.1;

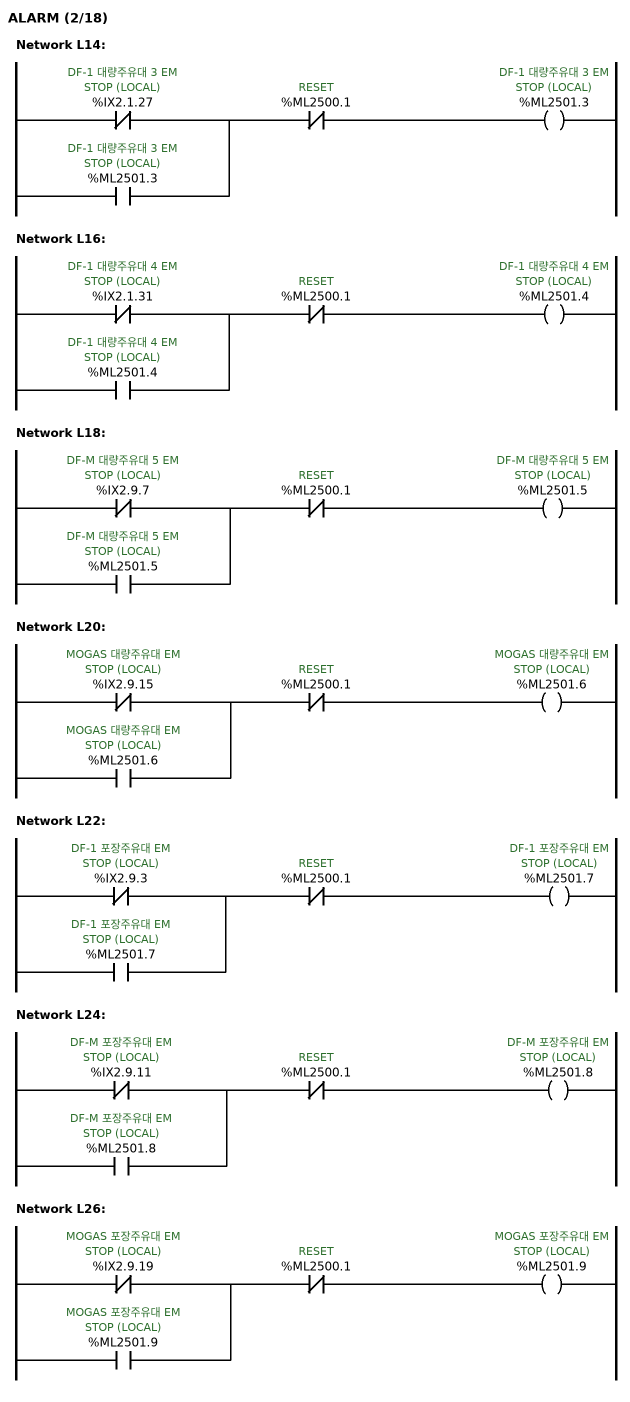
(* Rung L14 *)
%ML2501.3 := (NOT %IX2.1.27 OR %ML2501.3) AND NOT %ML2500.1;
(* Rung L16 *)
%ML2501.4 := (NOT %IX2.1.31 OR %ML2501.4) AND NOT %ML2500.1;
(* Rung L18 *)
%ML2501.5 := (NOT %IX2.9.7 OR %ML2501.5) AND NOT %ML2500.1;
(* Rung L20 *)
%ML2501.6 := (NOT %IX2.9.15 OR %ML2501.6) AND NOT %ML2500.1;
(* Rung L22 *)
%ML2501.7 := (NOT %IX2.9.3 OR %ML2501.7) AND NOT %ML2500.1;
(* Rung L24 *)
%ML2501.8 := (NOT %IX2.9.11 OR %ML2501.8) AND NOT %ML2500.1;
(* Rung L26 *)
%ML2501.9 := (NOT %IX2.9.19 OR %ML2501.9) AND NOT %ML2500.1;

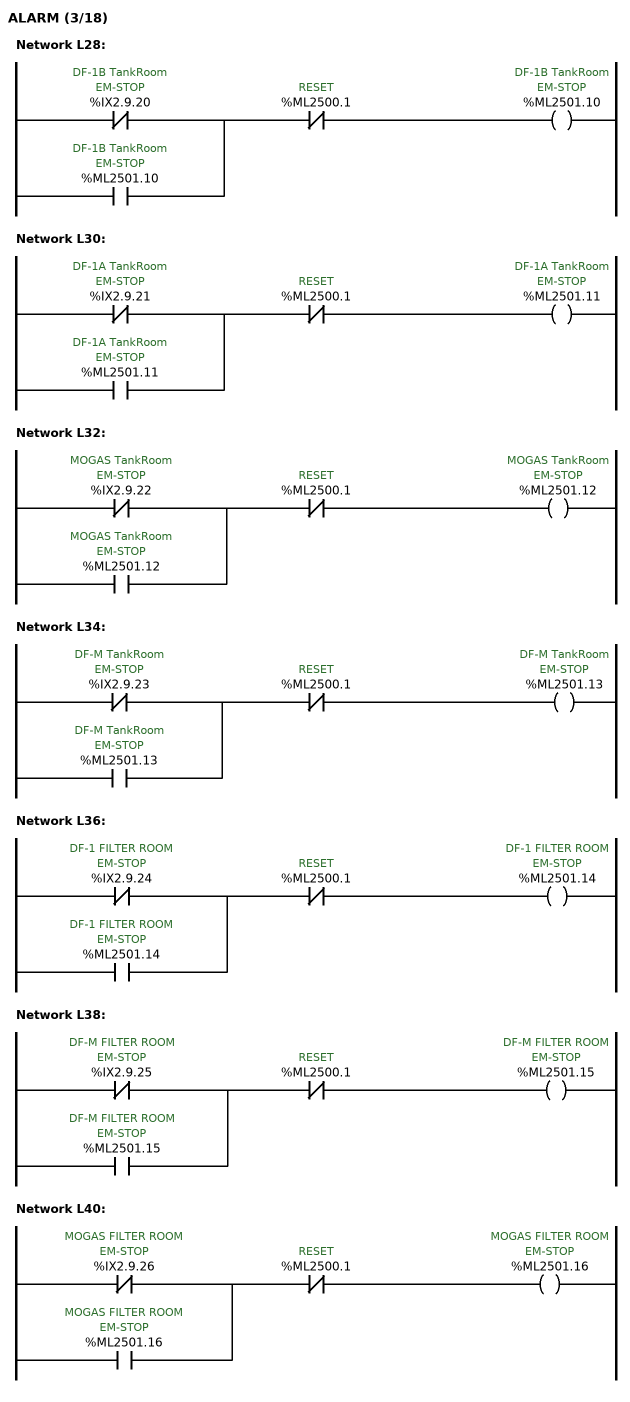
(* Rung L28 *)
%ML2501.10 := (NOT %IX2.9.20 OR %ML2501.10) AND NOT %ML2500.1;
(* Rung L30 *)
%ML2501.11 := (NOT %IX2.9.21 OR %ML2501.11) AND NOT %ML2500.1;
(* Rung L32 *)
%ML2501.12 := (NOT %IX2.9.22 OR %ML2501.12) AND NOT %ML2500.1;
(* Rung L34 *)
%ML2501.13 := (NOT %IX2.9.23 OR %ML2501.13) AND NOT %ML2500.1;
(* Rung L36 *)
%ML2501.14 := (NOT %IX2.9.24 OR %ML2501.14) AND NOT %ML2500.1;
(* Rung L38 *)
%ML2501.15 := (NOT %IX2.9.25 OR %ML2501.15) AND NOT %ML2500.1;
(* Rung L40 *)
%ML2501.16 := (NOT %IX2.9.26 OR %ML2501.16) AND NOT %ML2500.1;

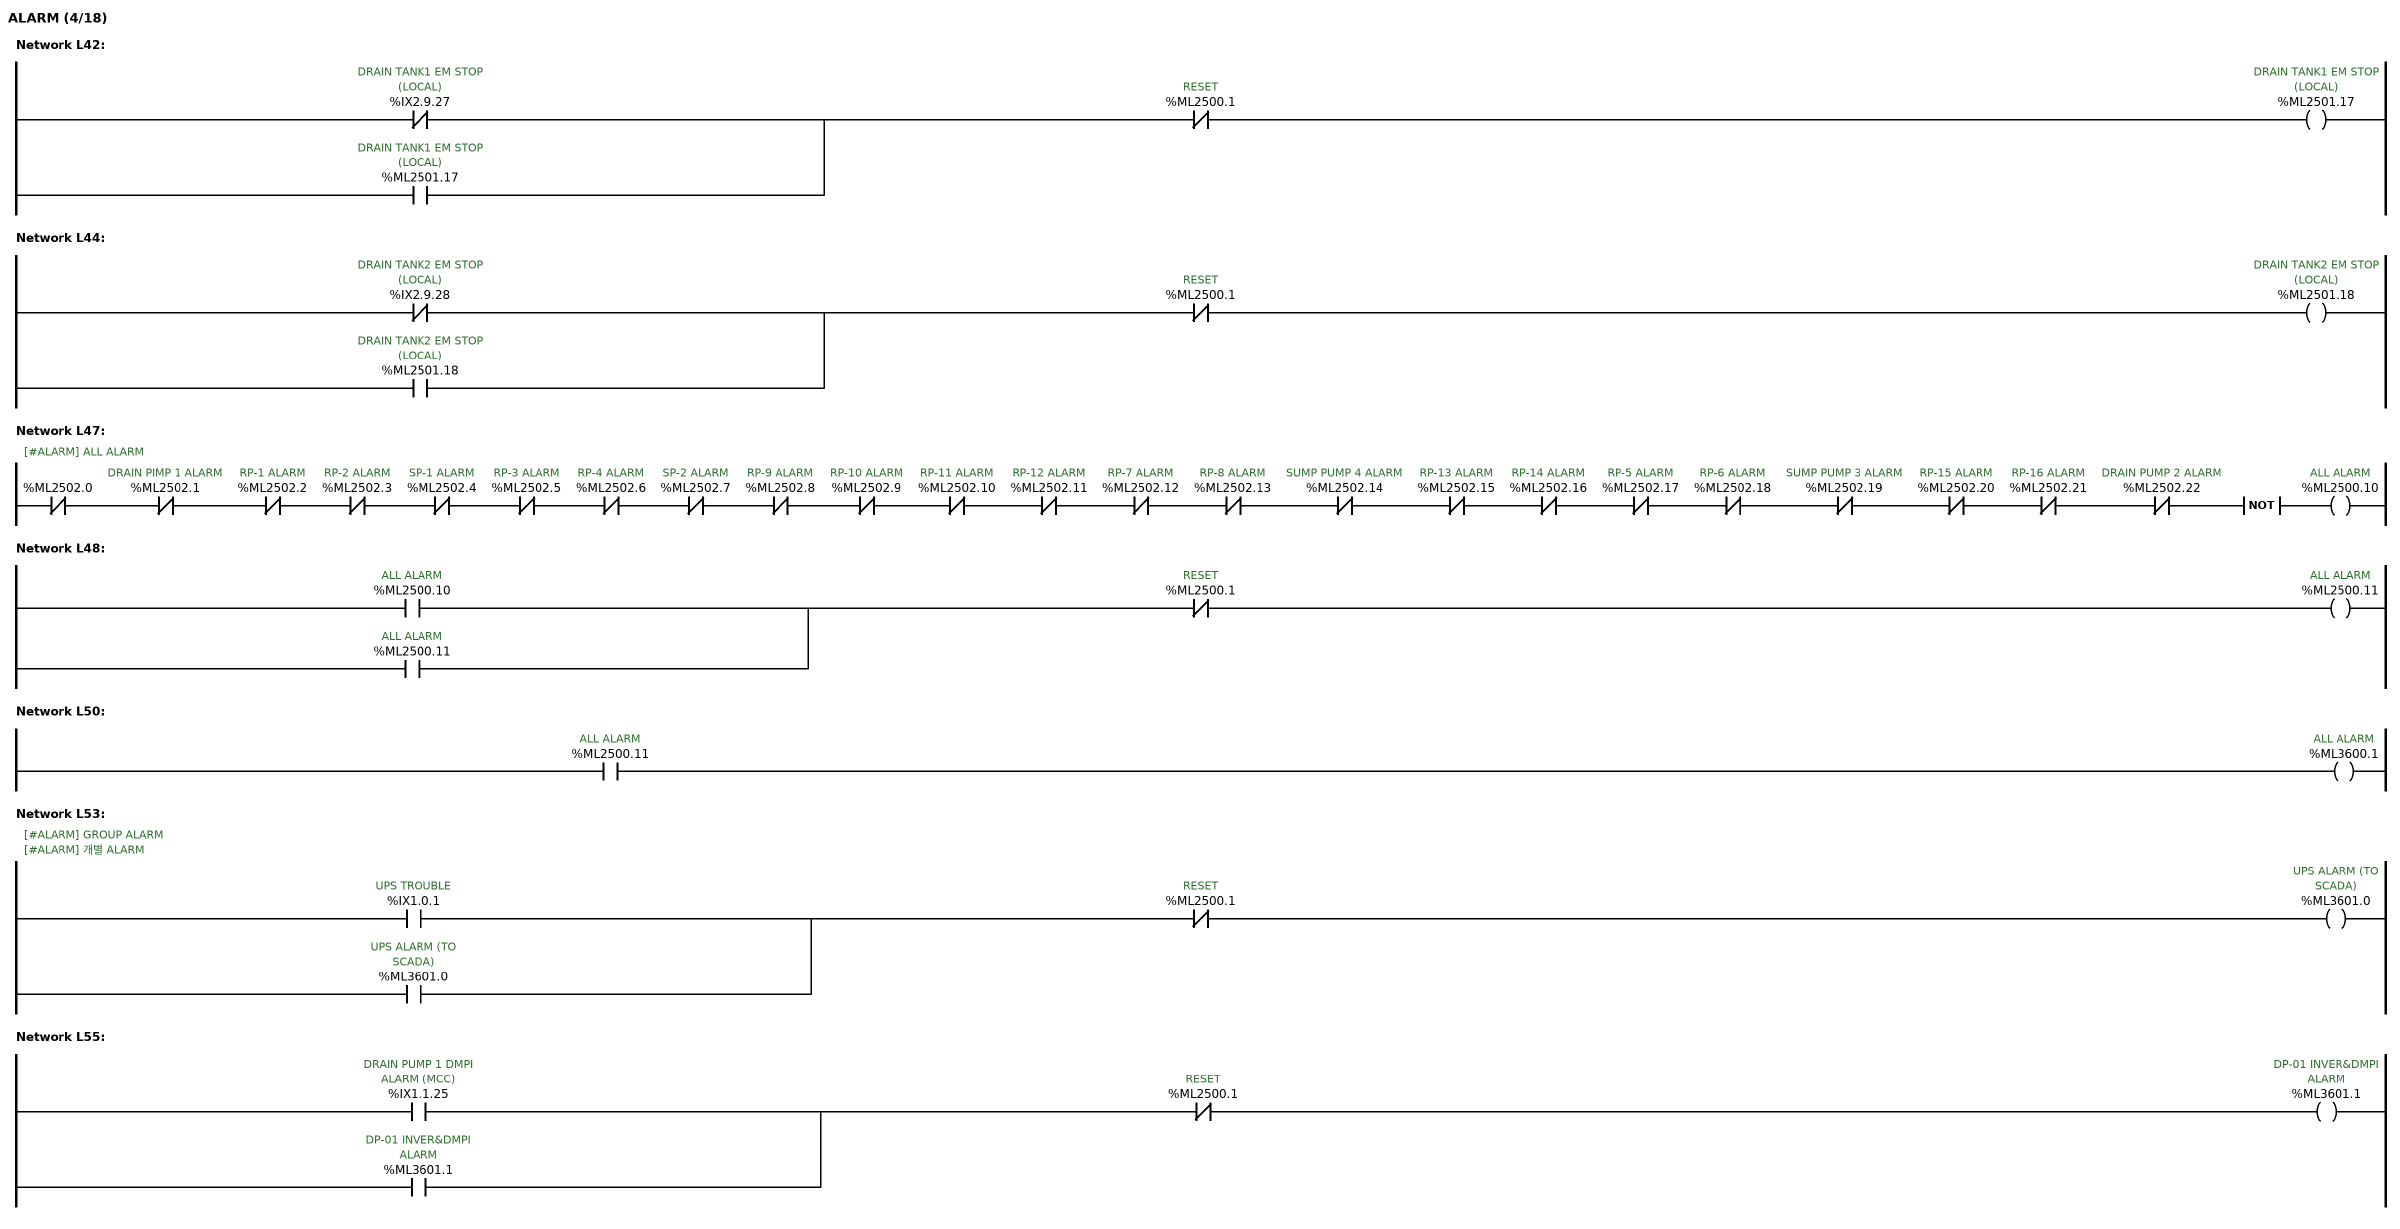
(* Rung L42 *)
%ML2501.17 := (NOT %IX2.9.27 OR %ML2501.17) AND NOT %ML2500.1;
(* Rung L44 *)
%ML2501.18 := (NOT %IX2.9.28 OR %ML2501.18) AND NOT %ML2500.1;
(* [#ALARM] ALL ALARM *)
(* Rung L47 *)
%ML2500.10 := NOT (NOT %ML2502.0 AND NOT %ML2502.1 AND NOT %ML2502.2 AND NOT %ML2502.3 AND NOT %ML2502.4 AND NOT %ML2502.5 AND NOT %ML2502.6 AND NOT %ML2502.7 AND NOT %ML2502.8 AND NOT %ML2502.9 AND NOT %ML2502.10 AND NOT %ML2502.11 AND NOT %ML2502.12 AND NOT %ML2502.13 AND NOT %ML2502.14 AND NOT %ML2502.15 AND NOT %ML2502.16 AND NOT %ML2502.17 AND NOT %ML2502.18 AND NOT %ML2502.19 AND NOT %ML2502.20 AND NOT %ML2502.21 AND NOT %ML2502.22);
(* Rung L48 *)
%ML2500.11 := (%ML2500.10 OR %ML2500.11) AND NOT %ML2500.1;
(* Rung L50 *)
%ML3600.1 := %ML2500.11;
(* [#ALARM] GROUP ALARM *)
(* [#ALARM] 개별 ALARM *)
(* Rung L53 *)
%ML3601.0 := (%IX1.0.1 OR %ML3601.0) AND NOT %ML2500.1;
(* Rung L55 *)
%ML3601.1 := (%IX1.1.25 OR %ML3601.1) AND NOT %ML2500.1;

